DATA_BLOCK "dbArchiveAutoShipping"
{ S7_Optimized_Access := 'TRUE' }
VERSION : 0.8
NON_RETAIN
"fbArchiveAutoShipping"

BEGIN

END_DATA_BLOCK

